PROGRAM MAIN
VAR
	fbAdd:		FB_1;
	fbMult:		FB_2;
	
	//New Fb
	fbDiv:		FB_Divide;
	
	nResult1:		INT;
	nResult2:		INT;
	nResult3:		INT;
END_VAR

fbAdd(nIn1:=10,
	  nIn2:=20,
	  nOut1=>nResult1);
	  
fbMult(nIn1:=10,
	  nIn2:=20,
	  nOut1=>nResult1);
	  
//New cool divide function
fbDiv(nDivIn1:=20,
	  nDivIn2:=10,
	  nDivOut=>nResult3);

END_PROGRAM

(* stored: Version 1.1.0.1, ProductVersion 3.1.4024.3
   POU MAIN: Id {00c6e621-0101-4866-bc50-1b8a8f77f956}, SpecialFunc None *)
